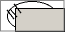
VISUALIZATION VISU_LAMPE  // 65x32
VAR_IN_OUT
	m_Input_ELMT_CHAUFF:	BLOCK_ELMT_CHAUFF;
END_VAR
    Ellipse (7,1 50x30), angle 331, colour toggle: m_Input_ELMT_CHAUFF.OUT_MCH
    Rectangle (15,8 50x24), angle 330
    Group (7,4 14x15), invisible if: NOT m_Input_ELMT_CHAUFF.OUT_MCH
        Line (7,15) (0,6)
        Line (10,13) (3,5)
        Line (14,9) (7,0)
END_VISUALIZATION

(* stored: Version 1.1.0.1, ProductVersion 3.1.4024.10
   Visu VISU_LAMPE: Id {444b16b0-1661-40c9-b6cc-8c4cca906c78} *)
